(* Logix 5000 project; controller Reto1_SeparatingEstation Emulate 5570 rev 30.12; software revision 30.00 *)

TASK MainTask (continuous, watchdog 500 ms) : MainProgram

MODULES
   Local : Emulate 5570 (ICP 2, rev 30.12)
      I_O : vendor 1 type 0 code 15 (ICP 3, rev 1.1, Output RPI 150 ms)
END_MODULES

VAR_GLOBAL   (* controller tags *)
   B_Verde : BOOL;
   Banda3 : BOOL;
   Bandera1 : BOOL := 1;
   Bandera2 : BOOL;
   GD_OUT_0 : BOOL := 1;
   GD_OUT_1 : BOOL;
   GD_OUT_2 : BOOL := 1;
   HMI_start : BOOL;
   Pusher_Azul : BOOL;
   Pusher_Verde : BOOL;
   Reset : TIMER;
   Sensor_Azul : BOOL;
   Sensor_paso1 : BOOL;
   Sensor_Verde : BOOL;
   start : BOOL;
   Stop : BOOL := 1;
   TimerB1 : TIMER := (PRE := 3000, ACC := 3000);
   TimerB2 : TIMER := (PRE := 1000, ACC := 1029);
   TimerPV : TIMER := (PRE := 4000, ACC := 4024);
   TimerPV2 : TIMER := (PRE := 2000);
   TimerV : TIMER := (PRE := 1500);
   TimerVerde : TIMER := (PRE := 2000, ACC := 2000);
   TimerVoff : TIMER := (PRE := 3000);
END_VAR

PROGRAM MainProgram   (* main routine MainRoutine *)

ROUTINE MainRoutine   (* ladder *)
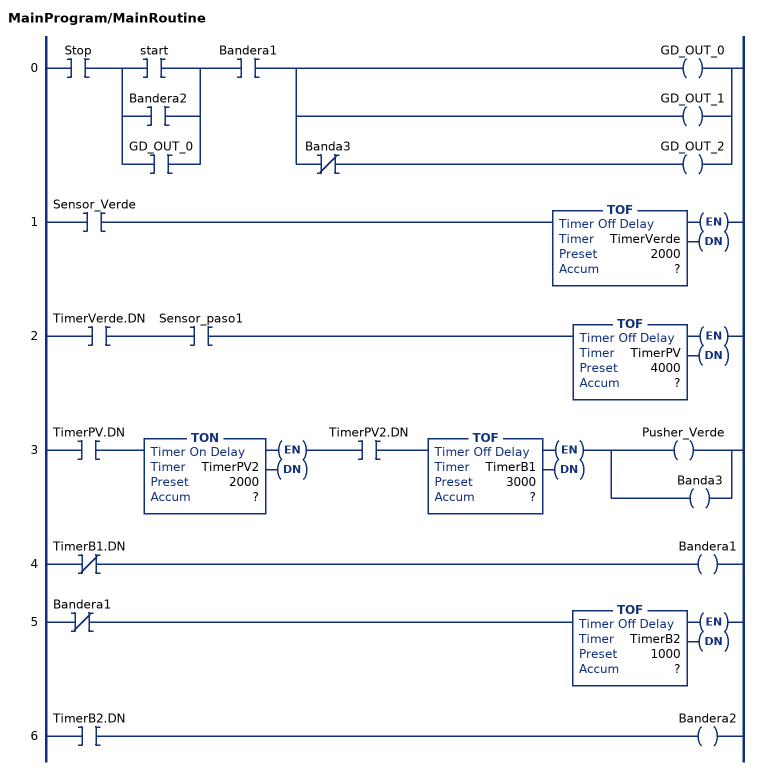
   0: XIC(Stop)[XIC(start) ,XIC(Bandera2) ,XIC(GD_OUT_0) ]XIC(Bandera1)[OTE(GD_OUT_0) ,OTE(GD_OUT_1) ,XIO(Banda3) OTE(GD_OUT_2) ];
   1: XIC(Sensor_Verde)TOF(TimerVerde,?,?);
   2: XIC(TimerVerde.DN)XIC(Sensor_paso1)TOF(TimerPV,?,?);
   3: XIC(TimerPV.DN)TON(TimerPV2,?,?)XIC(TimerPV2.DN)TOF(TimerB1,?,?)[OTE(Pusher_Verde) ,OTE(Banda3) ];
   4: XIO(TimerB1.DN)OTE(Bandera1);
   5: XIO(Bandera1)TOF(TimerB2,?,?);
   6: XIC(TimerB2.DN)OTE(Bandera2);
END_ROUTINE
END_PROGRAM
